{attribute 'GeneratedUsingTerminal: IL2302-B110-0016'}
{attribute addProperty BoxType "IL2302-B110-0016"}
{attribute addProperty Id "Term_23KL_D4CFBC220Term_394_Ix1000KL_8EF4D3E90"}
{attribute addProperty CRC "430890847"}
{attribute addProperty Size "0"}
{attribute addProperty Name "A_0023(IL2302-B110-0016)"}
TYPE A_0023_IL2302_B110_0016_19AEDF5F EXTENDS IL2302_A2FCADE7 :
STRUCT
	{attribute addProperty Name "Term_23"}
	Term_23 : KL_D4CFBC22;
	{attribute addProperty Name "Term_394_Ix1000"}
	Term_394_Ix1000 : KL_8EF4D3E9;
END_STRUCT
END_TYPE

(* stored: Version 1.2.0.0, ProductVersion 3.1.4024.11
   DUT A_0023_IL2302_B110_0016_19AEDF5F: Id {d21a49ac-db9a-4b22-96a6-62fe9d069728} *)
